Staubli VAL3: start.pgx

program start()
begin
      call prgm1()
end
